{attribute addProperty BoxType "EK1100-0000-0018"}
{attribute addProperty Id "Beckhoff_EL7xxxEK1122Beckhoff_EL7xxxEK1122_D459DE4F162A_0001_EL7031_0000_0016EL7031_4871A0C323229A_0002_EL7031_0000_0017EL7031_4871A0C323229A_0003_EL7031_0000_0018EL7031_6B71002F24030A_0004_EL7031_0000_0019EL7031_6B71002F24030A_0005_EL7031_0000_0020EL7031_6B71002F24030A_0006_EL7031_0000_0021EL7031_6B71002F24030A_0007_EL7031_0000_0022EL7031_6B71002F24030A_0008_EL7031_0000_0023EL7031_61C571CF24030A_0009_EL7031_0000_0024EL7031_61C571CF24030A_0010_EL7031_0000_0025EL7031_61C571CF24030A_0011_EL7031_0000_0026EL7031_61C571CF24030A_0012_EL7031_0030_0016EL7031_03DB887136846A_0013_EL7037_0000_0016EL7037_E93814AC24030A_0014_EL7037_0000_0017EL7037_E93814AC24030A_0015_EL7037_0000_0018EL7037_E93814AC24030A_0016_EL7037_0000_0019EL7037_E93814AC24030A_0017_EL7037_0000_0020EL7037_E93814AC24030A_0018_EL7041_0000_0016EL7041_204FAA6023229A_0019_EL7041_0000_0017EL7041_204FAA6023229A_0020_EL7041_0000_0018EL7041_034F0A8C24030A_0021_EL7041_0000_0019EL7041_034F0A8C24030A_0022_EL7041_0000_0020EL7041_034F0A8C24030A_0023_EL7041_0000_0021EL7041_034F0A8C24030A_0024_EL7041_0000_0022EL7041_034F0A8C24030A_0025_EL7041_0000_0023EL7041_D41ED1A824030A_0026_EL7041_0000_0024EL7041_D41ED1A824030A_0027_EL7041_0000_0025EL7041_D41ED1A824030A_0028_EL7041_0001_0016EL7041_43F8EB7626032.5A_0029_EL7041_0001_0017EL7041_41EBDE3723229A_0030_EL7041_0001_0018EL7041_62EB7EDB24030A_0031_EL7041_0001_0019EL7041_62EB7EDB24030A_0032_EL7041_0001_0020EL7041_62EB7EDB24030A_0033_EL7041_0001_0021EL7041_62EB7EDB24030A_0034_EL7041_0001_0022EL7041_11B2965424030A_0035_EL7041_0001_0023EL7041_11B2965424030A_0036_EL7041_0001_0024EL7041_11B2965424030A_0037_EL7041_0052_0016EL7041_61C571CF24030A_0038_EL7041_1000_0016EL7041_204FAA6023229A_0039_EL7041_1000_0017EL7041_204FAA6023229A_0040_EL7041_1000_0018EL7041_204FAA6023229A_0041_EL7041_1000_0019EL7041_204FAA6023229A_0042_EL7041_1000_0020EL7041_F71E714423229A_0043_EL7041_1000_0021EL7041_F71E714423229A_0044_EL7047_0000_0016EL7047_E93814AC24030A_0045_EL7047_0000_0017EL7047_E93814AC24030A_0046_EL7047_0000_0018EL7047_E93814AC24030A_0047_EL7047_0000_0019EL7047_E93814AC24030A_0048_EL7047_0000_0020EL7047_E93814AC24030A_0049_EL7047_0000_0021EL7047_E93814AC24030A_0050_EL7047_9014_0021EL7047_E93814AC24030A_0051_EL7411_0000_0016EL7411_5835FB8430438A_0052_EL7411_0000_0017EL7411_5835FB8430438A_0053_EL7411_0000_0018EL7411_5835FB8430438"}
{attribute addProperty CRC "623572225"}
{attribute addProperty SizeInBites "12988"}
{attribute addProperty SizeInBytes "1623.5"}
TYPE Beckhoff_EL7xxx_252AF501 EXTENDS EK1100_179A0949 :
STRUCT
	{attribute addProperty Name "Beckhoff_EL7xxxEK1122"}
	Beckhoff_EL7xxxEK1122 : Beckhoff_EL7xxxEK1122_D459DE4F;
	{attribute addProperty Name "A_0001_EL7031_0000_0016"}
	A_0001_EL7031_0000_0016 : EL7031_4871A0C3;
	{attribute addProperty Name "A_0002_EL7031_0000_0017"}
	A_0002_EL7031_0000_0017 : EL7031_4871A0C3;
	{attribute addProperty Name "A_0003_EL7031_0000_0018"}
	A_0003_EL7031_0000_0018 : EL7031_6B71002F;
	{attribute addProperty Name "A_0004_EL7031_0000_0019"}
	A_0004_EL7031_0000_0019 : EL7031_6B71002F;
	{attribute addProperty Name "A_0005_EL7031_0000_0020"}
	A_0005_EL7031_0000_0020 : EL7031_6B71002F;
	{attribute addProperty Name "A_0006_EL7031_0000_0021"}
	A_0006_EL7031_0000_0021 : EL7031_6B71002F;
	{attribute addProperty Name "A_0007_EL7031_0000_0022"}
	A_0007_EL7031_0000_0022 : EL7031_6B71002F;
	{attribute addProperty Name "A_0008_EL7031_0000_0023"}
	A_0008_EL7031_0000_0023 : EL7031_61C571CF;
	{attribute addProperty Name "A_0009_EL7031_0000_0024"}
	A_0009_EL7031_0000_0024 : EL7031_61C571CF;
	{attribute addProperty Name "A_0010_EL7031_0000_0025"}
	A_0010_EL7031_0000_0025 : EL7031_61C571CF;
	{attribute addProperty Name "A_0011_EL7031_0000_0026"}
	A_0011_EL7031_0000_0026 : EL7031_61C571CF;
	{attribute addProperty Name "A_0012_EL7031_0030_0016"}
	A_0012_EL7031_0030_0016 : EL7031_03DB8871;
	{attribute addProperty Name "A_0013_EL7037_0000_0016"}
	A_0013_EL7037_0000_0016 : EL7037_E93814AC;
	{attribute addProperty Name "A_0014_EL7037_0000_0017"}
	A_0014_EL7037_0000_0017 : EL7037_E93814AC;
	{attribute addProperty Name "A_0015_EL7037_0000_0018"}
	A_0015_EL7037_0000_0018 : EL7037_E93814AC;
	{attribute addProperty Name "A_0016_EL7037_0000_0019"}
	A_0016_EL7037_0000_0019 : EL7037_E93814AC;
	{attribute addProperty Name "A_0017_EL7037_0000_0020"}
	A_0017_EL7037_0000_0020 : EL7037_E93814AC;
	{attribute addProperty Name "A_0018_EL7041_0000_0016"}
	A_0018_EL7041_0000_0016 : EL7041_204FAA60;
	{attribute addProperty Name "A_0019_EL7041_0000_0017"}
	A_0019_EL7041_0000_0017 : EL7041_204FAA60;
	{attribute addProperty Name "A_0020_EL7041_0000_0018"}
	A_0020_EL7041_0000_0018 : EL7041_034F0A8C;
	{attribute addProperty Name "A_0021_EL7041_0000_0019"}
	A_0021_EL7041_0000_0019 : EL7041_034F0A8C;
	{attribute addProperty Name "A_0022_EL7041_0000_0020"}
	A_0022_EL7041_0000_0020 : EL7041_034F0A8C;
	{attribute addProperty Name "A_0023_EL7041_0000_0021"}
	A_0023_EL7041_0000_0021 : EL7041_034F0A8C;
	{attribute addProperty Name "A_0024_EL7041_0000_0022"}
	A_0024_EL7041_0000_0022 : EL7041_034F0A8C;
	{attribute addProperty Name "A_0025_EL7041_0000_0023"}
	A_0025_EL7041_0000_0023 : EL7041_D41ED1A8;
	{attribute addProperty Name "A_0026_EL7041_0000_0024"}
	A_0026_EL7041_0000_0024 : EL7041_D41ED1A8;
	{attribute addProperty Name "A_0027_EL7041_0000_0025"}
	A_0027_EL7041_0000_0025 : EL7041_D41ED1A8;
	{attribute addProperty Name "A_0028_EL7041_0001_0016"}
	A_0028_EL7041_0001_0016 : EL7041_43F8EB76;
	{attribute addProperty Name "A_0029_EL7041_0001_0017"}
	A_0029_EL7041_0001_0017 : EL7041_41EBDE37;
	{attribute addProperty Name "A_0030_EL7041_0001_0018"}
	A_0030_EL7041_0001_0018 : EL7041_62EB7EDB;
	{attribute addProperty Name "A_0031_EL7041_0001_0019"}
	A_0031_EL7041_0001_0019 : EL7041_62EB7EDB;
	{attribute addProperty Name "A_0032_EL7041_0001_0020"}
	A_0032_EL7041_0001_0020 : EL7041_62EB7EDB;
	{attribute addProperty Name "A_0033_EL7041_0001_0021"}
	A_0033_EL7041_0001_0021 : EL7041_62EB7EDB;
	{attribute addProperty Name "A_0034_EL7041_0001_0022"}
	A_0034_EL7041_0001_0022 : EL7041_11B29654;
	{attribute addProperty Name "A_0035_EL7041_0001_0023"}
	A_0035_EL7041_0001_0023 : EL7041_11B29654;
	{attribute addProperty Name "A_0036_EL7041_0001_0024"}
	A_0036_EL7041_0001_0024 : EL7041_11B29654;
	{attribute addProperty Name "A_0037_EL7041_0052_0016"}
	A_0037_EL7041_0052_0016 : EL7041_61C571CF;
	{attribute addProperty Name "A_0038_EL7041_1000_0016"}
	A_0038_EL7041_1000_0016 : EL7041_204FAA60;
	{attribute addProperty Name "A_0039_EL7041_1000_0017"}
	A_0039_EL7041_1000_0017 : EL7041_204FAA60;
	{attribute addProperty Name "A_0040_EL7041_1000_0018"}
	A_0040_EL7041_1000_0018 : EL7041_204FAA60;
	{attribute addProperty Name "A_0041_EL7041_1000_0019"}
	A_0041_EL7041_1000_0019 : EL7041_204FAA60;
	{attribute addProperty Name "A_0042_EL7041_1000_0020"}
	A_0042_EL7041_1000_0020 : EL7041_F71E7144;
	{attribute addProperty Name "A_0043_EL7041_1000_0021"}
	A_0043_EL7041_1000_0021 : EL7041_F71E7144;
	{attribute addProperty Name "A_0044_EL7047_0000_0016"}
	A_0044_EL7047_0000_0016 : EL7047_E93814AC;
	{attribute addProperty Name "A_0045_EL7047_0000_0017"}
	A_0045_EL7047_0000_0017 : EL7047_E93814AC;
	{attribute addProperty Name "A_0046_EL7047_0000_0018"}
	A_0046_EL7047_0000_0018 : EL7047_E93814AC;
	{attribute addProperty Name "A_0047_EL7047_0000_0019"}
	A_0047_EL7047_0000_0019 : EL7047_E93814AC;
	{attribute addProperty Name "A_0048_EL7047_0000_0020"}
	A_0048_EL7047_0000_0020 : EL7047_E93814AC;
	{attribute addProperty Name "A_0049_EL7047_0000_0021"}
	A_0049_EL7047_0000_0021 : EL7047_E93814AC;
	{attribute addProperty Name "A_0050_EL7047_9014_0021"}
	A_0050_EL7047_9014_0021 : EL7047_E93814AC;
	{attribute addProperty Name "A_0051_EL7411_0000_0016"}
	A_0051_EL7411_0000_0016 : EL7411_5835FB84;
	{attribute addProperty Name "A_0052_EL7411_0000_0017"}
	A_0052_EL7411_0000_0017 : EL7411_5835FB84;
	{attribute addProperty Name "A_0053_EL7411_0000_0018"}
	A_0053_EL7411_0000_0018 : EL7411_5835FB84;
END_STRUCT
END_TYPE

(* stored: Version 1.2.0.0, ProductVersion 3.1.4024.9
   DUT Beckhoff_EL7xxx_252AF501: Id {5b678528-305d-4005-8e48-ee81bfaa5bff} *)
